FUNCTION_BLOCK INTERNAL FB_State1 EXTENDS FB_State
VAR_INPUT
END_VAR
VAR_OUTPUT
END_VAR
VAR
END_VAR

END_FUNCTION_BLOCK

(* stored: Version 1.1.0.1, ProductVersion 3.1.4024.12
   POU FB_State1: Id {c4644caa-b43f-0f72-216e-6df04c9fdcfe}, SpecialFunc None *)
